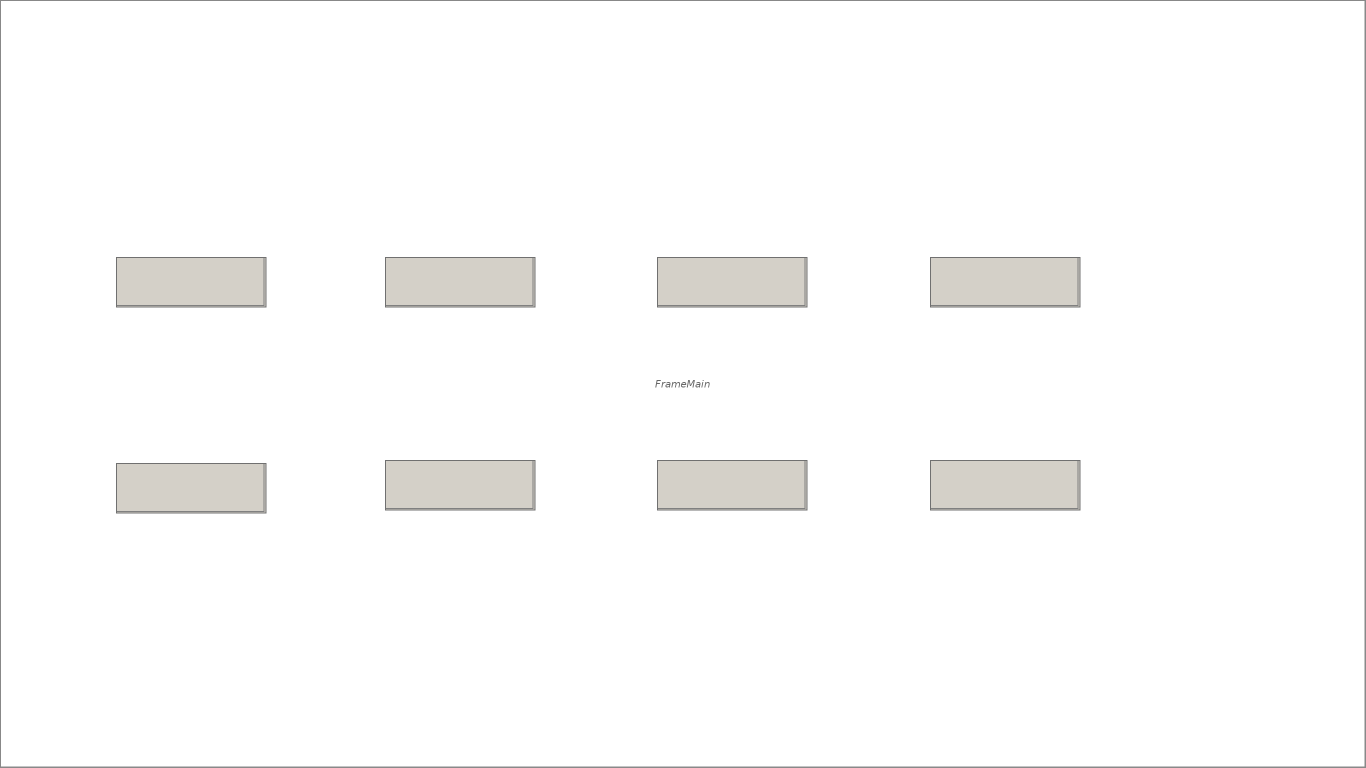
VISUALIZATION PageSetting  // 1366x768
    Frame (0,0 1366x768)
        shows FrameMain()
    Button (385,257 150x50), text list: 'StationName', text index: 1
        OnMouseClick: change screen: PageSetting_Steering
    Button (657,257 150x50), text list: 'StationName', text index: 2
        OnMouseClick: change screen: PageSetting_OpenLock
    Button (930,257 150x50), text list: 'StationName', text index: 3
        OnMouseClick: change screen: PageSetting_TakeUc
    Button (116,463 150x50), text list: 'StationName', text index: 4
        OnMouseClick: change screen: PageSetting_TakeUc_M
    Button (385,460 150x50), text list: 'StationName', text index: 5
        OnMouseClick: change screen: PageSetting_UnloadFrock
    Button (657,460 150x50), text list: 'StationName', text index: 6
        OnMouseClick: change screen: PageSetting_Unload_L
    Button (930,460 150x50), text list: 'StationName', text index: 7
        OnMouseClick: change screen: PageSetting_Other
    Button (116,257 150x50), text list: 'StationName', text index: 0
        OnMouseClick: change screen: PageSetting_AcquireLoad
END_VISUALIZATION

(* stored: Version 1.1.0.1, ProductVersion 3.1.4024.3
   Visu PageSetting: Id {529c123a-33c8-4230-9318-8d92f144d495} *)
